(*

short summary
=============

.. <legal notes>

legal notes
=================
| SPDX-FileCopyrightText: © 2023 ekvip automation GmbH <info@ekvip.de>
| SPDX-License-Identifier: Apache-2.0
| For details check: Apache-2.0_

.. _Apache-2.0: https://www.apache.org/licenses/LICENSE-2.0

.. </legal notes>

*)

{warning 'header is generated please add your documentation'}
{attribute 'qualified_only'}
VAR_GLOBAL CONSTANT
	SIZE_OF_CONTAINS_DATASET:USINT := 23;
END_VAR

VAR_GLOBAL
	containsDataSetCommon : ARRAY[0..SIZE_OF_CONTAINS_DATASET] OF containsDataStr := [
		// test number 0
		(	StringToTest		:= 'hello',
		  	WStringToTest 		:= "Hello",
			StringToContain 	:= 'h',
			WStringToContain	:= "h",
			IgnoreCases			:= TRUE,
			ExpectedResult  	:= FALSE,
			typeToTest      	:= TypeToTest.TEST_STRING	),
		
		// test number 1	
		(	StringToTest		:= 'hello',
		  	WStringToTest 		:= "Hello",
			StringToContain 	:= 'h',
			WStringToContain	:= "h",
			IgnoreCases			:= TRUE,
			ExpectedResult  	:= FALSE,
			typeToTest      	:= TypeToTest.TEST_WSTRING	),
		
		// test number 2		
		(	StringToTest		:= 'дивный новый мир',
		  	WStringToTest 		:= "дивный новый мир",
			StringToContain 	:= 'нов',
			WStringToContain	:= "нов",
			IgnoreCases			:= TRUE,
			ExpectedResult  	:= FALSE,
			typeToTest      	:= TypeToTest.TEST_WSTRING	),

		// test number 3				
		(	StringToTest		:= 'дивный новый мир',
		  	WStringToTest 		:= "дивный новый мир",
			StringToContain 	:= 'ноa',
			WStringToContain	:= "ноa",
			IgnoreCases			:= TRUE,
			ExpectedResult  	:= TRUE,
			typeToTest      	:= TypeToTest.TEST_WSTRING	),

		// test number 4				
		(	StringToTest		:= 'дивный новый мир',
		  	WStringToTest 		:= "дивный новый мир",
			StringToContain 	:= 'нов',
			WStringToContain	:= "нов",
			IgnoreCases			:= TRUE,
			ExpectedResult  	:= FALSE,
			typeToTest      	:= TypeToTest.TEST_STRING	),
	
		// test number 5			
		(	StringToTest		:= 'дивный новый мир',
		  	WStringToTest 		:= "дивный новый мир",
			StringToContain 	:= 'ноa',
			WStringToContain	:= "ноa",
			IgnoreCases			:= TRUE,
			ExpectedResult  	:= TRUE,
			typeToTest      	:= TypeToTest.TEST_STRING	),
			
		// test number 6			
		(	StringToTest		:= '',
		  	WStringToTest 		:= "",
			StringToContain 	:= ' ',
			WStringToContain	:= " ",
			IgnoreCases			:= TRUE,
			ExpectedResult  	:= TRUE,
			typeToTest      	:= TypeToTest.TEST_STRING	),
			
		// test number 7			
		(	StringToTest		:= '',
		  	WStringToTest 		:= "",
			StringToContain 	:= ' ',
			WStringToContain	:= " ",
			IgnoreCases			:= TRUE,
			ExpectedResult  	:= TRUE,
			typeToTest      	:= TypeToTest.TEST_WSTRING	),
			
		// test number 8			
		(	StringToTest		:= ' ',
		  	WStringToTest 		:= " ",
			StringToContain 	:= ' ',
			WStringToContain	:= " ",
			IgnoreCases			:= TRUE,
			ExpectedResult  	:= FALSE,
			typeToTest      	:= TypeToTest.TEST_STRING	),
			
		// test number 9			
		(	StringToTest		:= ' ',
		  	WStringToTest 		:= " ",
			StringToContain 	:= ' ',
			WStringToContain	:= " ",
			IgnoreCases			:= TRUE,
			ExpectedResult  	:= FALSE,
			typeToTest      	:= TypeToTest.TEST_WSTRING	),
			
		// test number 10			
		(	StringToTest		:= ' ',
		  	WStringToTest 		:= " ",
			StringToContain 	:= ' ',
			WStringToContain	:= " ",
			IgnoreCases			:= TRUE,
			ExpectedResult  	:= FALSE,
			typeToTest      	:= TypeToTest.TEST_STRING	),
			
		// test number 11			
		(	StringToTest		:= 'Brave new World',
		  	WStringToTest 		:= "Brave new World",
			StringToContain 	:= 'brave',
			WStringToContain	:= "brave",
			IgnoreCases			:= FALSE,
			ExpectedResult  	:= TRUE,
			typeToTest      	:= TypeToTest.TEST_WSTRING	),
			
		// test number 12			
		(	StringToTest		:= 'Brave new World',
		  	WStringToTest 		:= "Brave new World",
			StringToContain 	:= 'brave',
			WStringToContain	:= "brave",
			IgnoreCases			:= FALSE,
			ExpectedResult  	:= TRUE,
			typeToTest      	:= TypeToTest.TEST_WSTRING	),
			
		// test number 13			
		(	StringToTest		:= 'Brave new World',
		  	WStringToTest 		:= "Brave new World",
			StringToContain 	:= 'brave',
			WStringToContain	:= "brave",
			IgnoreCases			:= TRUE,
			ExpectedResult  	:= FALSE,
			typeToTest      	:= TypeToTest.TEST_WSTRING	),
			
		// test number 14			
		(	StringToTest		:= 'Brave new World',
		  	WStringToTest 		:= "Brave new World",
			StringToContain 	:= 'brave',
			WStringToContain	:= "brave",
			IgnoreCases			:= TRUE,
			ExpectedResult  	:= FALSE,
			typeToTest      	:= TypeToTest.TEST_WSTRING	),
			
		// test number 15			
		(	StringToTest		:= '²345',
		  	WStringToTest 		:= "²345",
			StringToContain 	:= '2',
			WStringToContain	:= "2",
			IgnoreCases			:= TRUE,
			ExpectedResult  	:= TRUE,
			typeToTest      	:= TypeToTest.TEST_STRING	),
			
		// test number 16			
		(	StringToTest		:= '2345',
		  	WStringToTest 		:= "²345",
			StringToContain 	:= '2',
			WStringToContain	:= "2",
			IgnoreCases			:= TRUE,
			ExpectedResult  	:= TRUE,
			typeToTest      	:= TypeToTest.TEST_WSTRING	),
			
		// test number 17			
		(	StringToTest		:= '²345',
		  	WStringToTest 		:= "²345",
			StringToContain 	:= '2',
			WStringToContain	:= "2",
			IgnoreCases			:= FALSE,
			ExpectedResult  	:= TRUE,
			typeToTest      	:= TypeToTest.TEST_STRING	),
			
		// test number 18			
		(	StringToTest		:= '²345',
		  	WStringToTest 		:= "²345",
			StringToContain 	:= '2',
			WStringToContain	:= "2",
			IgnoreCases			:= FALSE,
			ExpectedResult  	:= TRUE,
			typeToTest      	:= TypeToTest.TEST_WSTRING	),
			
		// test number 19			
		(	StringToTest		:= '',
		  	WStringToTest 		:= "👪",
			StringToContain 	:= '',
			WStringToContain	:= "👪",
			IgnoreCases			:= FALSE,
			ExpectedResult  	:= FALSE,
			typeToTest      	:= TypeToTest.TEST_WSTRING	),
			
		// test number 20			
		(	StringToTest		:= ' hello world ',
		  	WStringToTest 		:= " hello world ",
			StringToContain 	:= '  ',
			WStringToContain	:= "  ",
			IgnoreCases			:= FALSE,
			ExpectedResult  	:= TRUE,
			typeToTest      	:= TypeToTest.TEST_WSTRING	),
			
		// test number 21			
		(	StringToTest		:= ' hello world ',
		  	WStringToTest 		:= " hello world ",
			StringToContain 	:= '  ',
			WStringToContain	:= "  ",
			IgnoreCases			:= FALSE,
			ExpectedResult  	:= TRUE,
			typeToTest      	:= TypeToTest.TEST_STRING	),
			
		// test number 22			
		(	StringToTest		:= '',
		  	WStringToTest 		:= "∛",
			StringToContain 	:= '',
			WStringToContain	:= "√∛∜",
			IgnoreCases			:= FALSE,
			ExpectedResult  	:= TRUE,
			typeToTest      	:= TypeToTest.TEST_WSTRING	),
			
		// test number 23			
		(	StringToTest		:= '',
		  	WStringToTest 		:= "∭∝√∛∜",
			StringToContain 	:= '',
			WStringToContain	:= "∬",
			IgnoreCases			:= FALSE,
			ExpectedResult  	:= TRUE,
			typeToTest      	:= TypeToTest.TEST_WSTRING	)

					
						
	];
END_VAR

(* stored: Version 1.1.0.1, ProductVersion 3.1.4024.12
   GVL containsTestDataSet: Id {6d41b659-b9dc-43b2-9481-85491c9ce04f} *)
